// TIA Portal V20 export
TYPE "zd_SCS_ModeBox_OutputsLT"
// stored: Access Published, IsFailsafeCompliant true, Namespace Safety
   STRUCT
      SO1_Disabled : Bool;   // SAFE OUTPUT 1 DISABLED LT
      SO2_PendantReq : Bool;   // SAFE OUTPUT 2 PENDANT REQUIRED LT
      SO3_Spare : Bool;   // SAFE OUTPUT 3 SPARE NOT USE
   END_STRUCT;
END_TYPE
